// TIA Portal V20 export
TYPE "typeIdentRf"
// stored: Access Published
   STRUCT
      IdentRfAntena : Array[0.."NO_OF_RF_ANTENNA_DEVICES"] of "LSicar_typeIdentInterfaceHmi";
   END_STRUCT;
END_TYPE
